Staubli VAL3: AA_Chessie.dtx

frame fFrame = {x=374.8, y=3.07, z=-517.036829, rx=-180, fatherId=world[0]}
jointRx jCaseNoire = {j1=-5.017205, j2=92.568227, j3=85.506286, j4=-5.02125, j5=92.334481, j6=182.995856}
jointRx jDepart = {j1=20.811233, j2=126.617326, j3=-10.855704, j5=64.238378, j6=-69.188767}
jointRx jInitial
jointRx jStart = {j1=-4.35, j2=22.39, j3=131, j5=25.77, j6=50.65}
mdesc mDeplacement = {accel=250}
mdesc mDepose = {accel=25, vel=50}
mdesc mPrise = {accel=25, vel=50}
num nTESTSIO
num nX = 4
num nY = 9
num ncompteur[10]
num ni = 32
pointRx pCaseNoire[33]
  [0] = {x=374.8, y=3.07, z=-495.75, rx=-180, shoulder=lefty, elbow=epositive, wrist=wpositive, fatherId=world[0]}
  [1] = {x=430.4, y=3.07, z=-495.75, rx=-180, shoulder=lefty, elbow=epositive, wrist=wpositive, fatherId=world[0]}
  [2] = {x=486, y=3.07, z=-495.75, rx=-180, shoulder=lefty, elbow=epositive, wrist=wpositive, fatherId=world[0]}
  [3] = {x=541.6, y=3.07, z=-495.75, rx=-180, shoulder=lefty, elbow=epositive, wrist=wpositive, fatherId=world[0]}
  [4] = {x=402.6, y=30.87, z=-495.75, rx=-180, shoulder=lefty, elbow=epositive, wrist=wpositive, fatherId=world[0]}
  [5] = {x=458.2, y=30.87, z=-495.75, rx=-180, shoulder=lefty, elbow=epositive, wrist=wpositive, fatherId=world[0]}
  [6] = {x=513.8, y=30.87, z=-495.75, rx=-180, shoulder=lefty, elbow=epositive, wrist=wpositive, fatherId=world[0]}
  [7] = {x=569.4, y=30.87, z=-495.75, rx=-180, shoulder=lefty, elbow=epositive, wrist=wpositive, fatherId=world[0]}
  [8] = {x=374.8, y=58.67, z=-495.75, rx=-180, shoulder=lefty, elbow=epositive, wrist=wpositive, fatherId=world[0]}
  [9] = {x=430.4, y=58.67, z=-495.75, rx=-180, shoulder=lefty, elbow=epositive, wrist=wpositive, fatherId=world[0]}
  [10] = {x=486, y=58.67, z=-495.75, rx=-180, shoulder=lefty, elbow=epositive, wrist=wpositive, fatherId=world[0]}
  [11] = {x=541.6, y=58.67, z=-495.75, rx=-180, shoulder=lefty, elbow=epositive, wrist=wpositive, fatherId=world[0]}
  [12] = {x=402.6, y=86.47, z=-495.75, rx=-180, shoulder=lefty, elbow=epositive, wrist=wpositive, fatherId=world[0]}
  [13] = {x=458.2, y=86.47, z=-495.75, rx=-180, shoulder=lefty, elbow=epositive, wrist=wpositive, fatherId=world[0]}
  [14] = {x=513.8, y=86.47, z=-495.75, rx=-180, shoulder=lefty, elbow=epositive, wrist=wpositive, fatherId=world[0]}
  [15] = {x=569.4, y=86.47, z=-495.75, rx=-180, shoulder=lefty, elbow=epositive, wrist=wpositive, fatherId=world[0]}
  [16] = {x=374.8, y=114.27, z=-495.75, rx=-180, shoulder=lefty, elbow=epositive, wrist=wpositive, fatherId=world[0]}
  [17] = {x=430.4, y=114.27, z=-495.75, rx=-180, shoulder=lefty, elbow=epositive, wrist=wpositive, fatherId=world[0]}
  [18] = {x=486, y=114.27, z=-495.75, rx=-180, shoulder=lefty, elbow=epositive, wrist=wpositive, fatherId=world[0]}
  [19] = {x=541.6, y=114.27, z=-495.75, rx=-180, shoulder=lefty, elbow=epositive, wrist=wpositive, fatherId=world[0]}
  [20] = {x=402.6, y=142.07, z=-495.75, rx=-180, shoulder=lefty, elbow=epositive, wrist=wpositive, fatherId=world[0]}
  [21] = {x=458.2, y=142.07, z=-495.75, rx=-180, shoulder=lefty, elbow=epositive, wrist=wpositive, fatherId=world[0]}
  [22] = {x=513.8, y=142.07, z=-495.75, rx=-180, shoulder=lefty, elbow=epositive, wrist=wpositive, fatherId=world[0]}
  [23] = {x=569.4, y=142.07, z=-495.75, rx=-180, shoulder=lefty, elbow=epositive, wrist=wpositive, fatherId=world[0]}
  [24] = {x=374.8, y=169.87, z=-495.75, rx=-180, shoulder=lefty, elbow=epositive, wrist=wpositive, fatherId=world[0]}
  [25] = {x=430.4, y=169.87, z=-495.75, rx=-180, shoulder=lefty, elbow=epositive, wrist=wpositive, fatherId=world[0]}
  [26] = {x=486, y=169.87, z=-495.75, rx=-180, shoulder=lefty, elbow=epositive, wrist=wpositive, fatherId=world[0]}
  [27] = {x=541.6, y=169.87, z=-495.75, rx=-180, shoulder=lefty, elbow=epositive, wrist=wpositive, fatherId=world[0]}
  [28] = {x=402.6, y=197.67, z=-495.75, rx=-180, shoulder=lefty, elbow=epositive, wrist=wpositive, fatherId=world[0]}
  [29] = {x=458.2, y=197.67, z=-495.75, rx=-180, shoulder=lefty, elbow=epositive, wrist=wpositive, fatherId=world[0]}
  [30] = {x=513.8, y=197.67, z=-495.75, rx=-180, shoulder=lefty, elbow=epositive, wrist=wpositive, fatherId=world[0]}
  [31] = {x=569.4, y=197.67, z=-495.75, rx=-180, shoulder=lefty, elbow=epositive, wrist=wpositive, fatherId=world[0]}
  [32] = {fatherId=world[0]}
pointRx pPieceMangees[26]
  [0] = {x=374.8, y=-97.99178, z=-500.37, rx=-180, shoulder=lefty, elbow=epositive, wrist=wpositive, fatherId=world[0]}
  [1] = {x=394.8, y=-97.99178, z=-500.37, rx=-180, shoulder=lefty, elbow=epositive, wrist=wpositive, fatherId=world[0]}
  [2] = {x=414.8, y=-97.99178, z=-500.37, rx=-180, shoulder=lefty, elbow=epositive, wrist=wpositive, fatherId=world[0]}
  [3] = {x=434.8, y=-97.99178, z=-500.37, rx=-180, shoulder=lefty, elbow=epositive, wrist=wpositive, fatherId=world[0]}
  [4] = {x=454.8, y=-97.99178, z=-500.37, rx=-180, shoulder=lefty, elbow=epositive, wrist=wpositive, fatherId=world[0]}
  [5] = {x=474.8, y=-97.99178, z=-500.37, rx=-180, shoulder=lefty, elbow=epositive, wrist=wpositive, fatherId=world[0]}
  [6] = {x=374.8, y=-117.99178, z=-500.37, rx=-180, shoulder=lefty, elbow=epositive, wrist=wpositive, fatherId=world[0]}
  [7] = {x=394.8, y=-117.99178, z=-500.37, rx=-180, shoulder=lefty, elbow=epositive, wrist=wpositive, fatherId=world[0]}
  [8] = {x=414.8, y=-117.99178, z=-500.37, rx=-180, shoulder=lefty, elbow=epositive, wrist=wpositive, fatherId=world[0]}
  [9] = {x=434.8, y=-117.99178, z=-500.37, rx=-180, shoulder=lefty, elbow=epositive, wrist=wpositive, fatherId=world[0]}
  [10] = {x=454.8, y=-117.99178, z=-500.37, rx=-180, shoulder=lefty, elbow=epositive, wrist=wpositive, fatherId=world[0]}
  [11] = {x=474.8, y=-117.99178, z=-500.37, rx=-180, shoulder=lefty, elbow=epositive, wrist=wpositive, fatherId=world[0]}
  [12] = {x=374.8, y=-137.99178, z=-500.37, rx=-180, shoulder=lefty, elbow=epositive, wrist=wpositive, fatherId=world[0]}
  [13] = {x=394.8, y=-137.99178, z=-500.37, rx=-180, shoulder=lefty, elbow=epositive, wrist=wpositive, fatherId=world[0]}
  [14] = {x=414.8, y=-137.99178, z=-500.37, rx=-180, shoulder=lefty, elbow=epositive, wrist=wpositive, fatherId=world[0]}
  [15] = {x=434.8, y=-137.99178, z=-500.37, rx=-180, shoulder=lefty, elbow=epositive, wrist=wpositive, fatherId=world[0]}
  [16] = {x=454.8, y=-137.99178, z=-500.37, rx=-180, shoulder=lefty, elbow=epositive, wrist=wpositive, fatherId=world[0]}
  [17] = {x=474.8, y=-137.99178, z=-500.37, rx=-180, shoulder=lefty, elbow=epositive, wrist=wpositive, fatherId=world[0]}
  [18] = {x=374.8, y=-157.99178, z=-500.37, rx=-180, shoulder=lefty, elbow=epositive, wrist=wpositive, fatherId=world[0]}
  [19] = {x=394.8, y=-157.99178, z=-500.37, rx=-180, shoulder=lefty, elbow=epositive, wrist=wpositive, fatherId=world[0]}
  [20] = {x=414.8, y=-157.99178, z=-500.37, rx=-180, shoulder=lefty, elbow=epositive, wrist=wpositive, fatherId=world[0]}
  [21] = {x=434.8, y=-157.99178, z=-500.37, rx=-180, shoulder=lefty, elbow=epositive, wrist=wpositive, fatherId=world[0]}
  [22] = {x=454.8, y=-157.99178, z=-500.37, rx=-180, shoulder=lefty, elbow=epositive, wrist=wpositive, fatherId=world[0]}
  [23] = {x=474.8, y=-157.99178, z=-500.37, rx=-180, shoulder=lefty, elbow=epositive, wrist=wpositive, fatherId=world[0]}
  [24] = {x=374.8, y=-177.99178, z=-500.37, rx=-180, shoulder=lefty, elbow=epositive, wrist=wpositive, fatherId=world[0]}
  [25] = {x=394.8, y=-177.99178, z=-500.37, rx=-180, shoulder=lefty, elbow=epositive, wrist=wpositive, fatherId=world[0]}
pointRx pTable = {fatherId=fFrame[0]}
public sio sData = {link=Socket\staubli_server}
tool tTool = {x=63.134763, y=38.954373, z=16.017439, rx=-90.869915, ry=61.402378, rz=90.763801, fatherId=flange[0], ioLink=valve1}
trsf trAppro = {z=-40}
string sString[2]
  [0] = "nTESTIO"
  [1] = "nTESTIO"
